% RSLogix 500 project SECUENCIA DE PISTONES.RSS, saved by version 8.40.00.08 %
PROJECT "UNTITLED"    % processor: Bul.1763 MicroLogix 1100 Series A %

PROGRAM FILES
  LAD 2   9 rungs
  LAD 3   2 rungs

DATA FILES
  O0 OUTPUT  4 elements
  I1 INPUT  6 elements
  S2 STATUS  66 elements
  B3 BINARY  1 elements
  T4 TIMER  1 elements
  C5 COUNTER  1 elements
  R6 CONTROL  1 elements
  N7 INTEGER  1 elements
  F8 FLOAT  1 elements

LADDER 2
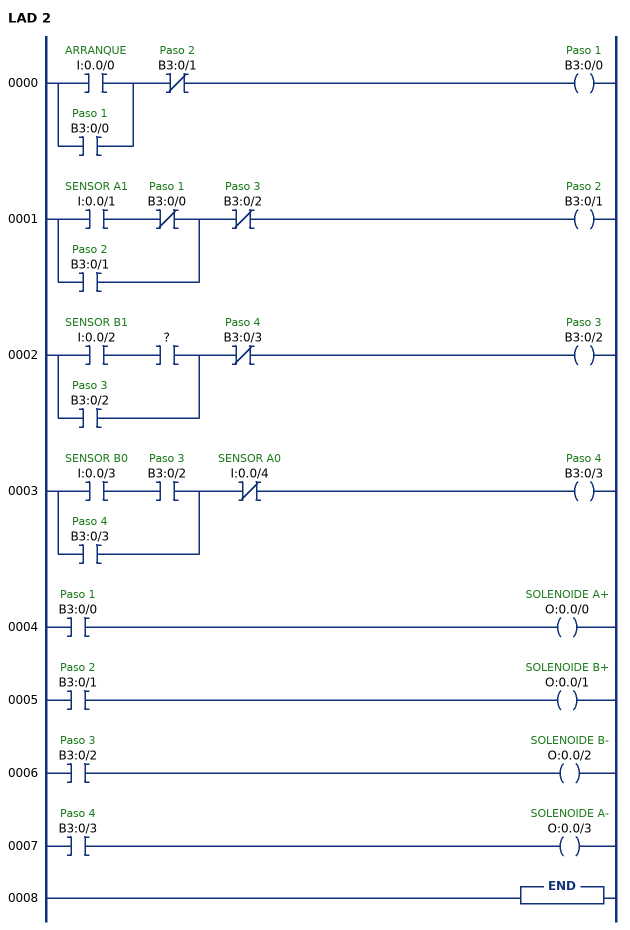
% Rung: 0 %
SOR BST XIC I:0.0/0 NXB XIC B3:0/0 BND XIO B3:0/1 OTE B3:0/0 EOR
%   I:0.0/0  "ARRANQUE" %
%   B3:0/0  "Paso 1" %
%   B3:0/1  "Paso 2" %
% Rung: 1 %
SOR BST XIC I:0.0/1 XIO B3:0/0 NXB XIC B3:0/1 BND XIO B3:0/2 OTE B3:0/1 EOR
%   I:0.0/1  "SENSOR A1" %
%   B3:0/0  "Paso 1" %
%   B3:0/1  "Paso 2" %
%   B3:0/2  "Paso 3" %
% Rung: 2 %  % edit flag set %
SOR BST XIC I:0.0/2 XIC ? NXB XIC B3:0/2 BND XIO B3:0/3 OTE B3:0/2 EOR
%   I:0.0/2  "SENSOR B1" %
%   B3:0/2  "Paso 3" %
%   B3:0/3  "Paso 4" %
% Rung: 3 %
SOR BST XIC I:0.0/3 XIC B3:0/2 NXB XIC B3:0/3 BND XIO I:0.0/4 OTE B3:0/3 EOR
%   I:0.0/3  "SENSOR B0" %
%   B3:0/2  "Paso 3" %
%   B3:0/3  "Paso 4" %
%   I:0.0/4  "SENSOR A0" %
% Rung: 4 %
SOR XIC B3:0/0 OTE O:0.0/0 EOR
%   B3:0/0  "Paso 1" %
%   O:0.0/0  "SOLENOIDE A+" %
% Rung: 5 %
SOR XIC B3:0/1 OTE O:0.0/1 EOR
%   B3:0/1  "Paso 2" %
%   O:0.0/1  "SOLENOIDE B+" %
% Rung: 6 %
SOR XIC B3:0/2 OTE O:0.0/2 EOR
%   B3:0/2  "Paso 3" %
%   O:0.0/2  "SOLENOIDE B-" %
% Rung: 7 %
SOR XIC B3:0/3 OTE O:0.0/3 EOR
%   B3:0/3  "Paso 4" %
%   O:0.0/3  "SOLENOIDE A-" %
% Rung: 8 %
SOR END EOR

LADDER 3
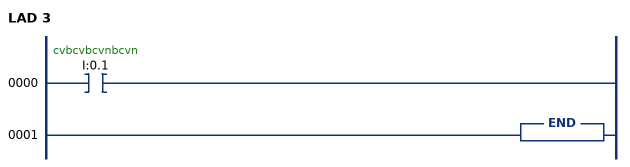
% Rung: 0 %  % edit flag set %
SOR XIC I:0.1 EOR
%   I:0.1  "cvbcvbcvnbcvn" %
% Rung: 1 %
SOR END EOR

OTHER DOCUMENTED ADDRESSES
  I  
  I:0.0/5  TR  "aa"
